INTERFACE ITcoSelector EXTENDS ITcoState

METHOD RequestState
VAR_INPUT
	State : INT;
END_VAR
END_METHOD

END_INTERFACE

(* stored: Version 1.1.0.1
   Itf ITcoSelector: Id {8b8caf52-afbd-4335-9286-252c4dc67aa2}
   Method RequestState: Id {447295ce-7b18-4f8f-a16f-4797226f59b0} *)
